{attribute addProperty BoxType "EL2252--0000"}
{attribute addProperty Id "StartTimeAT %Q*UDINT324"}
{attribute addProperty CRC "1998329195"}
{attribute addProperty SizeInBites "32"}
{attribute addProperty SizeInBytes "4"}
TYPE DC_Sync_Start_771C156B :
STRUCT
	{attribute addProperty Name "StartTime"}
	StartTime AT %Q* : UDINT;
END_STRUCT
END_TYPE

(* stored: Version 1.2.0.0, ProductVersion 3.1.4024.9
   DUT DC_Sync_Start_771C156B: Id {c6340f2e-e883-4bc1-9f52-b89a9ff7621b} *)
